{attribute 'qualified_only'}
{attribute "to_string'}
TYPE E_CommandList :
(
	ERR := -1,
	NULL := 0,
	LIST,
	HOM,
	SCAN,
	MTP,
	MOVA,
	MOVR,
	STAT,
	CALIB,
	PARAM
);
END_TYPE
//  ERR = '-1'

(* stored: Version 1.1.0.1, ProductVersion 3.1.4024.12
   EnumerationTextList E_CommandList: Id {7c9f0e93-a341-4256-b328-6006ed70ad3e} *)
